// TwinCAT 3 PLC project PLC
// ProgramVersion: 3.1.4024.0
// libraries:
//   Tc2_Standard, * (Beckhoff Automation GmbH)
//   Tc2_System, * (Beckhoff Automation GmbH)
//   Tc3_Module, * (Beckhoff Automation GmbH)
//   Util, * (System)
// project tree:
//   Diagnostic/ GVL_Diagnostic.TcGVL, ST_Diagnostic.TcDUT
//   FSM/Coordinator/Enums/ E_FSM_Step.TcTLEO
//   FSM/Coordinator/FBs/ FB_FSM.TcPOU, FB_FSM_Diagnostic.TcPOU, FB_FSM_ReadCmd.TcPOU, FB_FSM_ReadCtrl.TcPOU, FB_FSM_ReadInputs.TcPOU, FB_FSM_WriteOutputs.TcPOU
//   FSM/Coordinator/ FB_FSM_Main.TcPOU
//   FSM/Coordinator/FCs/ FC_AllError.TcPOU, FC_AllStopped.TcPOU
//   FSM/Coordinator/Structs/ ST_FSM_Cmd.TcDUT, ST_FSM_Ctrl.TcDUT, ST_FSM_In.TcDUT, ST_FSM_Out.TcDUT, ST_FSM_Params.TcDUT, ST_FSM_RawIn.TcDUT, ST_FSM_RawOut.TcDUT, ST_FSM_Status.TcDUT
//   FSM/Z1/ E_Z1_Step.TcTLEO, FB_Z1_FSM.TcPOU, ST_Z1_Params.TcDUT, ST_Z1_Status.TcDUT
//   FSM/Z2/ E_Z2_Step.TcTLEO, FB_Z2_FSM.TcPOU, ST_Z2_Params.TcDUT, ST_Z2_Status.TcDUT
//   FSM/Z3/ E_Z3_Step.TcTLEO, FB_Z3_FSM.TcPOU, ST_Z3_Params.TcDUT, ST_Z3_Status.TcDUT
//   FSM/Z4/ E_Z4_Step.TcTLEO, FB_Z4_FSM.TcPOU, ST_Z4_Params.TcDUT, ST_Z4_Status.TcDUT
//   FSM/Z5/ E_Z5_Step.TcTLEO, FB_Z5_FSM.TcPOU, ST_Z5_Params.TcDUT, ST_Z5_Status.TcDUT
//   FSM/Z6/ E_Z6_Step.TcTLEO, FB_Z6_FSM.TcPOU, ST_Z6_Params.TcDUT, ST_Z6_Status.TcDUT
//   / PlcTask.TcTTO (not stored)
//   POUs/ MAIN.TcPOU
// real-time tasks:
//   TASK PlcTask: cycle T#10ms, priority 20, ADS port 350
// motion (NC):
// I/O:
//   DEVICE Dispositivo 1 (EtherCAT)
//   DEVICE Dispositivo 4 (EtherCAT), AmsNetId 5.85.198.60.5.1
//     Terminale 10 (EK1100)
// variable links:
//   PLC Instance <-> Device 4 (EtherCAT)/Term 10 (EK1100)/Term 11 (EL1809)
//     PlcTask Inputs/MAIN.stRawIn.bAckButton <-> Channel 12/Input
//     PlcTask Inputs/MAIN.stRawIn.bEmergency <-> Channel 13/Input
//     PlcTask Inputs/MAIN.stRawIn.bI{1..9} <-> Channel {1..9}/Input  (9 links)
//     PlcTask Inputs/MAIN.stRawIn.bStartButton <-> Channel 10/Input
//     PlcTask Inputs/MAIN.stRawIn.bStopButton <-> Channel 11/Input
//   PLC Instance <-> Device 4 (EtherCAT)/Term 10 (EK1100)/Term 12 (EL2809)
//     PlcTask Outputs/MAIN.stRawOut.bGreen <-> Channel 11/Output
//     PlcTask Outputs/MAIN.stRawOut.bQ{1..10} <-> Channel {1..10}/Output  (10 links)
//     PlcTask Outputs/MAIN.stRawOut.bRed <-> Channel 12/Output
//     PlcTask Outputs/MAIN.stRawOut.bYellow <-> Channel 13/Output

// ---- Diagnostic/ST_Diagnostic.TcDUT
TYPE ST_Diagnostic :
STRUCT
	aCritical : ARRAY[0..GVL_Diagnostic.cMAXEVENTS - 1] OF BOOL;	// eventi critici
	aError : ARRAY[0..GVL_Diagnostic.cMAXEVENTS - 1] OF BOOL;		// errori
	aWarning : ARRAY[0..GVL_Diagnostic.cMAXEVENTS - 1] OF BOOL;		// segnalazioni
	aInfo : ARRAY[0..GVL_Diagnostic.cMAXEVENTS - 1] OF BOOL;		// informazioni
	aVerbose : ARRAY[0..GVL_Diagnostic.cMAXEVENTS - 1] OF BOOL;		// messaggi
END_STRUCT
END_TYPE

// ---- FSM/Coordinator/Enums/E_FSM_Step.TcTLEO
{attribute 'qualified_only'}
{attribute 'strict'}
TYPE E_FSM_Step :
(
	(* special steps *)
	NoStep := -32767,		// nessuno step
	Unknown := -32000,		// step sconosciuto
	
	(* Error steps *)
	NeOrError := -990,		// non abilitata o in errore
	Recovering := -980,		// azzeramento errori

	(* Stop *)
	Stop := 0,				// stop
	
	(* Cycle *)
	Running := 100,			// funzionamento nominale delle zone
		
	(* Stopping *)
	Stopping := 900			// fase di arresto
);
END_TYPE
//  NoStep = '-32767'
//  Unknown = '-32000'
//  NeOrError = '-990'
//  Recovering = '-980'

// ---- FSM/Coordinator/Structs/ST_FSM_Cmd.TcDUT
TYPE ST_FSM_Cmd :
STRUCT
	bAck				:	BOOL;	(* Riconoscimento allarmi *)
	bStop				:	BOOL;	(* Arresta la macchina *)
	bStart				:	BOOL;	(* Mette in marcia la macchina *)
END_STRUCT
END_TYPE

// ---- FSM/Coordinator/Structs/ST_FSM_Ctrl.TcDUT
TYPE ST_FSM_Ctrl :
STRUCT
	bEmergency	:	BOOL;		// Emergenza. Deve essere TRUE perchè la macchina possa operare
	bEnable		:	BOOL;		// Abilitazione macchina. Deve essere TRUE perchè la macchina possa operare
END_STRUCT
END_TYPE

// ---- FSM/Coordinator/Structs/ST_FSM_In.TcDUT
TYPE ST_FSM_In :
STRUCT
	(* digital *)
	bEmergency		:	BOOL;				// emergenza (NC)
	bStartButton	:	BOOL;				// pulsante di start (NO)
	bStopButton		:	BOOL;				// pulsante di stop (NO)
	bAckButton		:	BOOL;				// pulsante di riconoscimento allarmi (NO)
	bI1				:	BOOL;				// Fine corsa anteriore slider 1 (NO)
	bI2				:	BOOL;				// Fine corsa posteriore slider 1 (NO)
	bI3				:	BOOL;				// Fine corsa anteriore slider 2 (NO)
	bI4				:	BOOL;				// Fine corsa posteriore slider 2 (NO)
	bI5				:	BOOL;				// Sensore ingresso slider 1 (NO)
	bI6				:	BOOL;				// Sensore presenza pezzo sotto la fresa (NO)	
	bI7				:	BOOL;				// Sensore presenza pezzo su nastro caricamento (ingresso) (NO)
	bI8				:	BOOL;				// Sensore presenza pezzo sotto il trapano (NO)
	bI9				:	BOOL;				// Sensore presenza pezzo su nastro di uscita (NO)
	
	(* analog *)

	
END_STRUCT
END_TYPE

// ---- FSM/Coordinator/Structs/ST_FSM_Out.TcDUT
TYPE ST_FSM_Out :
STRUCT
	bFixedYellow	:	BOOL;		// luce gialla fissa
	bBlinkingYellow	:	BOOL;		// luce gialla lampeggiante
	bFixedGreen		:	BOOL;		// luce verde fissa
	bBlinkingGreen	:	BOOL;		// luce verde lampeggiante	
	bFixedRed		:	BOOL;		// luce rossa fissa
	bBlinkingRed	:	BOOL;		// luce rossa lampeggiante	
	bQ1				:	BOOL;		// Rientro slider 1
	bQ2				:	BOOL;		// Estensione slider 1
	bQ3				:	BOOL;		// Rientro slider 2
	bQ4				:	BOOL;		// Estensione slider 2
	bQ5				:	BOOL;		// Motore nastro caricamento (ingresso zona Z1)
	bQ6				:	BOOL;		// Motore nastro zona fresa (Z3)
	bQ7				:	BOOL;		// Motore fresa
	bQ8				:	BOOL;		// Motore nastro zona trapano (Z4)
	bQ9				:	BOOL;		// Motore trapano
	bQ10			:	BOOL;		// Motore nastro scarico (uscita zona Z6)	
		
END_STRUCT
END_TYPE

// ---- FSM/Coordinator/Structs/ST_FSM_Params.TcDUT
TYPE ST_FSM_Params :
STRUCT
	tStoppingDelay	:	TIME	:=	T#2S;
END_STRUCT
END_TYPE

// ---- FSM/Coordinator/Structs/ST_FSM_RawIn.TcDUT
TYPE ST_FSM_RawIn :
STRUCT
	(* digital *)
	bEmergency		AT %I*	:	BOOL;		// emergenza (NC)
	bStartButton	AT %I*	:	BOOL;		// pulsante di start (NO)
	bStopButton		AT %I*	:	BOOL;		// pulsante di stop (NC)
	bAckButton		AT %I*	:	BOOL;		// pulsante di riconoscimento allarmi (NO)
	bI1				AT %I*	:	BOOL;		// Fine corsa anteriore slider 1 (NO)
	bI2				AT %I*	:	BOOL;		// Fine corsa posteriore slider 1 (NO)
	bI3				AT %I*	:	BOOL;		// Fine corsa anteriore slider 2 (NO)
	bI4				AT %I*	:	BOOL;		// Fine corsa posteriore slider 2 (NO)
	bI5				AT %I*	:	BOOL;		// Sensore ingresso slider 1 (NC)
	bI6				AT %I*	:	BOOL;		// Sensore presenza pezzo sotto la fresa (NC)	
	bI7				AT %I*	:	BOOL;		// Sensore presenza pezzo su nastro caricamento (ingresso) (NC)
	bI8				AT %I*	:	BOOL;		// Sensore presenza pezzo sotto il trapano (NC)
	bI9				AT %I*	:	BOOL;		// Sensore presenza pezzo su nastro di uscita (NC)
	
	(* analog *)

		
END_STRUCT
END_TYPE

// ---- FSM/Coordinator/Structs/ST_FSM_RawOut.TcDUT
TYPE ST_FSM_RawOut :
STRUCT
	bYellow		AT %Q*	:	BOOL;		// luce gialla
	bGreen		AT %Q*	:	BOOL;		// luce verde
	bRed		AT %Q*	:	BOOL;		// luce rossa	
	bQ1			AT %Q*	:	BOOL;		// Rientro slider 1
	bQ2			AT %Q*	:	BOOL;		// Estensione slider 1
	bQ3			AT %Q*	:	BOOL;		// Rientro slider 2
	bQ4			AT %Q*	:	BOOL;		// Estensione slider 2
	bQ5			AT %Q*	:	BOOL;		// Motore nastro caricamento (ingresso zona Z1)
	bQ6			AT %Q*	:	BOOL;		// Motore nastro zona fresa (Z3)
	bQ7			AT %Q*	:	BOOL;		// Motore fresa
	bQ8			AT %Q*	:	BOOL;		// Motore nastro zona trapano (Z4)
	bQ9			AT %Q*	:	BOOL;		// Motore trapano
	bQ10		AT %Q*	:	BOOL;		// Motore nastro scarico (uscita zona Z6)	
END_STRUCT
END_TYPE

// ---- FSM/Coordinator/Structs/ST_FSM_Status.TcDUT
TYPE ST_FSM_Status :
STRUCT
	bCritical	: BOOL;					// la macchina ha almento una condizione critica attiva
	bError		: BOOL;					// la macchina ha almento una condizione di errore attiva	
	bWarning	: BOOL;					// la macchina ha almeno una segnalazione attiva	
	bInfo		: BOOL;					// la macchina ha almeno una informazione attiva			
	bVerbose	: BOOL;					// la macchina ha almeno un messaggio attiva
	
	bFailure	: BOOL;					// la macchina è in avaria (critica + error)	
	eStep		: E_FSM_Step;			// passo della macchina a stati
	strStep		: STRING;				// passo come stringa
	tStepTime	: TIME;					// tempo di permanenza nel passo
	eErrorStep	: E_FSM_Step;			// passo in cui si è generato l'errore
	nErrorID	: DINT;					// codice di errore
	
	stZ1		: ST_Z1_Status;			// stato del dispositivo Z1
	stZ2		: ST_Z2_Status;			// stato del dispositivo Z2	
	stZ3		: ST_Z3_Status;			// stato del dispositivo Z3
	stZ4		: ST_Z4_Status;			// stato del dispositivo Z4	
	stZ5		: ST_Z5_Status;			// stato del dispositivo Z5
	stZ6		: ST_Z6_Status;			// stato del dispositivo Z6
END_STRUCT
END_TYPE

// ---- FSM/Z1/E_Z1_Step.TcTLEO
{attribute 'qualified_only'}
{attribute 'strict'}
TYPE E_Z1_Step :
(
	(* special steps *)
	NoStep := -32767,		// nessuno step
	Unknown := -32000,		// step sconosciuto
	
	(* Error steps *)
	NeOrError := -990,		// non abilitata o in errore
	Recovering := -980,		// azzeramento errori
		
	(* Stop *)
	Stop := 0,				// S0, stop
	
	(* Cycle *)
	Ready := 100,			// S1, pronto a ricevere pezzo
	DelayToFeeding := 120,	// S2, ritardo prima dell'avvio del nastro
	Loading := 140,			// S3, trasferimento pezzo verso Z2 
	DelayToZ2 := 160,		// S4, ritardo post sensore I5 verso Z2

	Done := 800,			// Ciclo concluso
	
	(* Stopping *)
	Stopping := 900	
);
END_TYPE
//  NoStep = '-32767'
//  Unknown = '-32000'
//  NeOrError = '-990'
//  Recovering = '-980'

// ---- FSM/Z1/ST_Z1_Params.TcDUT
TYPE ST_Z1_Params :
STRUCT
	tWaiting	:	TIME	:= T#3S;	// durata della fase di carico nuovo pezzo
	tTravelTime	:	TIME	:= T#4S;	// tempo per arrivare a I5
	tDelayToZ2	:	TIME	:= T#2S;	// ritardo per arrivare a Z2
	tStopDelay	:	TIME	:= T#1S;	// permanenza nello stato Stop
END_STRUCT
END_TYPE

// ---- FSM/Z1/ST_Z1_Status.TcDUT
TYPE ST_Z1_Status :
STRUCT
	eStep		:	E_Z1_Step;		// passo della macchina a stati per Z1
	strStep		:	STRING;			// passo come stringa
	tStepTime	:	TIME;			// tempo di permanenza nello stato
	eErrorStep	:	E_Z1_Step;		// stato in cui si è generato l'errore
	nErrorId	:	UDINT;			// id errore
END_STRUCT
END_TYPE

// ---- FSM/Z2/E_Z2_Step.TcTLEO
{attribute 'qualified_only'}
{attribute 'strict'}
TYPE E_Z2_Step :
(
	(* special steps *)
	NoStep := -32767,		// nessuno step
	Unknown := -32000,		// step sconosciuto
	
	(* Error steps *)
	NeOrError := -990,		// non abilitata o in errore
	Recovering := -980,		// azzeramento errori
		
	(* Stop *)
	Stop := 0,				// S0, stop
	
	(* Cycle *)
	Ready := 100,			// S1, pronto a ricevere pezzo
	WaitZ3Ready := 120,		// S2, aspetta che Z3 sia libera
	MoveForward := 140,		// S3, trasferimento pezzo verso Z2 
	MoveBackward := 160,	// S4, ritorno slitta

	Done := 800,			// Ciclo concluso
	
	(* Stopping *)
	Stopping := 900	
);
END_TYPE
//  NoStep = '-32767'
//  Unknown = '-32000'
//  NeOrError = '-990'
//  Recovering = '-980'

// ---- FSM/Z2/ST_Z2_Params.TcDUT
TYPE ST_Z2_Params :
STRUCT
	tMoving		:	TIME	:= T#6S;	// durata della fase di trasporto
	tStopDelay	:	TIME	:= T#1S;	// permanenza nello stato Stop
END_STRUCT
END_TYPE

// ---- FSM/Z2/ST_Z2_Status.TcDUT
TYPE ST_Z2_Status :
STRUCT
	eStep		:	E_Z2_Step;		// passo della macchina a stati per Z2
	strStep		:	STRING;			// passo come stringa
	tStepTime	:	TIME;			// tempo di permanenza nello stato
	eErrorStep	:	E_Z2_Step;		// stato in cui si è generato l'errore
	nErrorId	:	UDINT;			// id errore
	
END_STRUCT
END_TYPE

// ---- FSM/Z3/E_Z3_Step.TcTLEO
{attribute 'qualified_only'}
{attribute 'strict'}
TYPE E_Z3_Step :
(
	(* special steps *)
	NoStep := -32767,		// nessuno step
	Unknown := -32000,		// step sconosciuto
	
	(* Error steps *)
	NeOrError := -990,		// non abilitata o in errore
	Recovering := -980,		// azzeramento errori
		
	(* Stop *)
	Stop := 0,				// S0, stop
	
	(* Cycle *)
	Ready := 100,			// S1, pronto a ricevere pezzo
	MoveToMill := 120,		// S2, avanza il nastro fino alla fresa
	Milling := 140,			// S3, lavorazione con la fresa
	WaitZ4Ready := 160,		// S4, attende che Z4 sia ready
	MoveToZ4 := 180,		// S5, avanza il nastro fino a Z4

	Done := 800,			// Ciclo concluso
	
	(* Stopping *)
	Stopping := 900	
);
END_TYPE
//  NoStep = '-32767'
//  Unknown = '-32000'
//  NeOrError = '-990'
//  Recovering = '-980'

// ---- FSM/Z3/ST_Z3_Params.TcDUT
TYPE ST_Z3_Params :
STRUCT
	tMilling	:	TIME	:= T#6S;	// durata della fase di fresatura
	tDelayToZ4	:	TIME	:= T#3S;	// ritardo per arrivare a Z4
	tStopDelay	:	TIME	:= T#1S;	// permanenza nello stato Stop
	tRecovering	: TIME		:= T#2S; 	// tempo di uscita dallo stato di Recovering
END_STRUCT
END_TYPE

// ---- FSM/Z3/ST_Z3_Status.TcDUT
TYPE ST_Z3_Status :
STRUCT
	eStep		:	E_Z3_Step;		// passo della macchina a stati per Z3
	strStep		:	STRING;			// passo come stringa
	tStepTime	:	TIME;			// tempo di permanenza nello stato
	eErrorStep	:	E_Z3_Step;		// stato in cui si è generato l'errore
	nErrorId	:	UDINT;			// id errore
END_STRUCT
END_TYPE

// ---- FSM/Z4/E_Z4_Step.TcTLEO
{attribute 'qualified_only'}
{attribute 'strict'}
TYPE E_Z4_Step :
(
	(* special steps *)
	NoStep := -32767,		// nessuno step
	Unknown := -32000,		// step sconosciuto
	
	(* Error steps *)
	NeOrError := -990,		// non abilitata o in errore
	Recovering := -980,		// azzeramento errori
		
	(* Stop *)
	Stop := 0,				// S0, stop
	
	(* Cycle *)
	Ready := 100,			// S1, pronto a ricevere pezzo
	MoveToDrill := 120,		// S2, avanza il nastro fino al trapano
	Drilling := 140,		// S3, lavorazione con il trapano
	WaitZ5Ready := 160,		// S4, attende che Z5 sia ready
	MoveToZ5 := 180,		// S5, avanza il nastro fino a Z5

	Done := 800,			// Ciclo concluso
	
	(* Stopping *)
	Stopping := 900	
);
END_TYPE
//  NoStep = '-32767'
//  Unknown = '-32000'
//  NeOrError = '-990'
//  Recovering = '-980'

// ---- FSM/Z4/ST_Z4_Params.TcDUT
TYPE ST_Z4_Params :
STRUCT
	tDrilling	:	TIME	:= T#4S;	// durata della fase di foratura
	tDelayToZ5	:	TIME	:= T#1S;	// ritardo per arrivare a Z5
	tStopDelay	:	TIME	:= T#1S;	// permanenza nello stato Stop
	tRecovering :   TIME	:= T#2S;
END_STRUCT
END_TYPE

// ---- FSM/Z4/ST_Z4_Status.TcDUT
TYPE ST_Z4_Status :
STRUCT
	eStep		:	E_Z4_Step;		// passo della macchina a stati per Z4
	strStep		:	STRING;			// passo come stringa
	tStepTime	:	TIME;			// tempo di permanenza nello stato
	eErrorStep	:	E_Z4_Step;		// stato in cui si è generato l'errore
	nErrorId	:	UDINT;			// id errore
END_STRUCT
END_TYPE

// ---- FSM/Z5/E_Z5_Step.TcTLEO
{attribute 'qualified_only'}
{attribute 'strict'}
TYPE E_Z5_Step :
(
	(* special steps *)
	NoStep := -32767,		// nessuno step
	Unknown := -32000,		// step sconosciuto
	
	(* Error steps *)
	NeOrError := -990,		// non abilitata o in errore
	Recovering := -980,		// azzeramento errori
		
	(* Stop *)
	Stop := 0,				// S0, stop
	
	(* Cycle *)
	Ready := 100,			// S1, pronto a ricevere pezzo
	WaitZ6Ready := 120,		// S2, aspetta che Z6 sia libera
	MoveForward := 140,		// S3, trasferimento pezzo verso Z6 
	MoveBackward := 160,	// S4, ritorno slitta

	Done := 800,			// Ciclo concluso
	
	(* Stopping *)
	Stopping := 900	
);
END_TYPE
//  NoStep = '-32767'
//  Unknown = '-32000'
//  NeOrError = '-990'
//  Recovering = '-980'

// ---- FSM/Z5/ST_Z5_Params.TcDUT
TYPE ST_Z5_Params :
STRUCT
	tMoving		:	TIME	:= T#6S;	// durata della fase di trasporto
	tStopDelay	:	TIME	:= T#1S;	// permanenza nello stato Stop
END_STRUCT
END_TYPE

// ---- FSM/Z5/ST_Z5_Status.TcDUT
TYPE ST_Z5_Status :
STRUCT
	eStep		:	E_Z5_Step;		// passo della macchina a stati per Z5
	strStep		:	STRING;			// passo come stringa
	tStepTime	:	TIME;			// tempo di permanenza nello stato
	eErrorStep	:	E_Z5_Step;		// stato in cui si è generato l'errore
	nErrorId	:	UDINT;			// id errore
END_STRUCT
END_TYPE

// ---- FSM/Z6/E_Z6_Step.TcTLEO
{attribute 'qualified_only'}
{attribute 'strict'}
TYPE E_Z6_Step :
(
	(* special steps *)
	NoStep := -32767,		// nessuno step
	Unknown := -32000,		// step sconosciuto
	
	(* Error steps *)
	NeOrError := -990,		// non abilitata o in errore
	Recovering := -980,		// azzeramento errori
		
	(* Stop *)
	Stop := 0,				// S0, stop
	
	(* Cycle *)
	Ready := 100,			// S1, pronto a ricevere pezzo
	Loading := 120,			// S2, trasferimento pezzo verso I9
	WaitUnloading := 140,	// S3, attesa rimozione pezzo da piattaforma scarico 

	Done := 800,			// Ciclo concluso
	
	(* Stopping *)
	Stopping := 900	
);
END_TYPE
//  NoStep = '-32767'
//  Unknown = '-32000'
//  NeOrError = '-990'
//  Recovering = '-980'

// ---- FSM/Z6/ST_Z6_Params.TcDUT
TYPE ST_Z6_Params :
STRUCT
	tDelayToEnd	:	TIME	:= T#2S;	// ritardo per arrivare a fine nastro
	tUnloading	:	TIME	:= T#3S;	// durata della fase di scarico
	tStopDelay	:	TIME	:= T#1S;	// permanenza nello stato Stop
END_STRUCT
END_TYPE

// ---- FSM/Z6/ST_Z6_Status.TcDUT
TYPE ST_Z6_Status :
STRUCT
	eStep		:	E_Z6_Step;		// passo della macchina a stati per Z6
	strStep		:	STRING;			// passo come stringa
	tStepTime	:	TIME;			// tempo di permanenza nello stato
	eErrorStep	:	E_Z6_Step;		// stato in cui si è generato l'errore
	nErrorId	:	UDINT;			// id errore
END_STRUCT
END_TYPE

// ---- Diagnostic/GVL_Diagnostic.TcGVL
{attribute 'qualified_only'}
VAR_GLOBAL CONSTANT
	cMAXEVENTS : UDINT := 64;
END_VAR

// ---- FSM/Coordinator/FBs/FB_FSM.TcPOU
FUNCTION_BLOCK FB_FSM
VAR_INPUT
	stIn		:	ST_FSM_In;
	stCtrl		:	ST_FSM_Ctrl;
	stCmd		:	ST_FSM_Cmd;
	stParams	:	ST_FSM_Params;
END_VAR
VAR_IN_OUT
	stStatus	:	ST_FSM_Status;	
END_VAR
VAR_OUTPUT	
	eStep		:	E_FSM_Step;
	tStepTime	:	TIME;
	eErrStep	:	E_FSM_Step;
	nErrId		:	DINT;
	// Digital Outputs
	stOut		:	ST_FSM_Out;	
	
END_VAR
VAR
	// FSM internal variables
	bInitialized	:	BOOL;
	eNewstep		:	E_FSM_Step;
	bEntryact		:	BOOL;
	fbTonStep		:	TON;

	(* filters on other input from plant *)
	
	(* stop request *)	
	bStopRequest	:	BOOL;
	
	// all zones are stopped
	bAllZoneStopped	:	BOOL;	
END_VAR

IF NOT bInitialized THEN
	(* here you can wait events from other controllers *)
	eNewStep := E_FSM_Step.NoStep;
	stStatus.eStep := E_FSM_Step.NeOrError;
	bEntryact := FALSE;
	bInitialized := TRUE;
ELSE
	// --- FSM Cyclical Code ----------------------------------------------
	
	// update of the enabling conditions (bStop, alarms, etc.)
	
	// 1. FSM Preamble ----------------------------------------------------
    // 1.a State machine disabled or failure
	IF NOT stCtrl.bEnable OR NOT stCtrl.bEmergency OR stStatus.bFailure THEN
		eNewStep := E_FSM_Step.NeOrError;
	END_IF

	// 1.b Update eStep with the required step to perform
	//     and set bEntryact to FALSE in order to enable the Entry action
	IF eNewstep <> E_FSM_Step.NoStep THEN
		stStatus.eStep := eNewstep;
		eNewstep := E_FSM_Step.NoStep;
		bEntryact := FALSE;
	END_IF;	
	
	// 1.c Do filters on signals	

	
	// Do requests, for example to stop the machine
	IF stCmd.bStop THEN
		bStopRequest := TRUE;
	END_IF

	// 2. The main switch-case ---------------------------------------------------
	CASE stStatus.eStep OF
    E_FSM_Step.NeOrError :
			// on entry action
			IF NOT bEntryact THEN
				stStatus.bFailure := TRUE;
				bEntryact := TRUE;
			END_IF
			
			// body
			stOut.bFixedGreen := TRUE;
			stOut.bBlinkingGreen := FALSE;
			stOut.bFixedRed := FALSE;
			stOut.bBlinkingRed := FALSE;
			stOut.bFixedYellow := FALSE;
			stOut.bBlinkingYellow := FALSE;
					
			
			// next state transition
			IF stCtrl.bEnable THEN
				IF stCmd.bAck THEN
					eNewStep := E_Z3_Step.Recovering;
				END_IF
			END_IF
		
			// on exit action
			IF eNewStep <> E_Z3_Step.NoStep THEN
				nErrId := 0;
				eErrStep := E_Z3_Step.NoStep;
			END_IF
						
	ELSE
		// this happens also if we forget to code one step 
		eNewstep := E_FSM_Step.NeOrError;
		stStatus.eErrorStep := E_FSM_Step.Unknown;
		stStatus.nErrorID := -9;
	END_CASE;
	
	// 3. FSM Epilogue ------------------------------------------------------
	
	// Elapsed time into the current step
	fbTonStep(IN := (eNewstep = E_FSM_Step.NoStep), PT := T#500H );
	stStatus.tStepTime := fbTonStep.ET;
	
END_IF

END_FUNCTION_BLOCK

// ---- FSM/Coordinator/FBs/FB_FSM_Diagnostic.TcPOU
FUNCTION_BLOCK FB_FSM_Diagnostic
VAR_INPUT
	stIn : ST_FSM_In;
	stOut : ST_FSM_Out;
	stParams : ST_FSM_Params;
	stCtrl : ST_FSM_Ctrl;
	bHwError : BOOL;
	bAck : BOOL;
	stStatus : ST_FSM_Status;	
END_VAR
VAR_IN_OUT
END_VAR
VAR_OUTPUT
	bCritical	: BOOL;
	bError		: BOOL;
	bWarning	: BOOL;
	bInfo		: BOOL;
	bVerbose	: BOOL;
	bFailure	: BOOL;
	bBlinking	: BOOL;
	bFixed		: BOOL;
END_VAR
VAR
END_VAR

// on Ack, reset holding conditions
IF bAck THEN
	bCritical := FALSE;
	bError := FALSE;
	bWarning := FALSE;
	bInfo := FALSE;
	bVerbose := FALSE;
	bBlinking := FALSE;
END_IF

// update critical condition
bCritical := FC_AllError(stStatus) OR NOT stCtrl.bEmergency;

// update holding conditions
bFailure := bCritical OR bError;

bBlinking := bFailure;
bFixed := bWarning;

END_FUNCTION_BLOCK

// ---- FSM/Coordinator/FCs/FC_AllError.TcPOU
FUNCTION FC_AllError : BOOL
VAR_INPUT
	stStatus	:	ST_FSM_Status;
END_VAR
VAR
END_VAR

FC_AllError := (stStatus.stZ1.eStep = E_Z1_Step.NeOrError) AND
                 (stStatus.stZ2.eStep = E_Z2_Step.NeOrError) AND
                 (stStatus.stZ3.eStep = E_Z3_Step.NeOrError) AND	
                 (stStatus.stZ4.eStep = E_Z4_Step.NeOrError) AND
                 (stStatus.stZ5.eStep = E_Z5_Step.NeOrError) AND	
                 (stStatus.stZ6.eStep = E_Z6_Step.NeOrError);

END_FUNCTION

// ---- FSM/Coordinator/FBs/FB_FSM_ReadCmd.TcPOU
FUNCTION_BLOCK FB_FSM_ReadCmd
VAR_INPUT
	stIn	:	ST_FSM_In;
END_VAR
VAR_OUTPUT
	stCmd	:	ST_FSM_Cmd;
END_VAR
VAR
	fbTpStart	: TP;
	fbTpStop	: TP;	
	fbTpAck		: TP;
END_VAR

// filters on input button
fbTpStart( IN := stIn.bStartButton, PT := T#50MS );
fbTpStop( IN := stIn.bStopButton, PT := T#50MS );
fbTpAck( IN := stIn.bAckButton, PT := T#50MS );

stCmd.bStart	:= fbTpStart.Q;
stCmd.bStop		:= fbTpStop.Q;
stCmd.bAck		:= fbTpAck.Q;

END_FUNCTION_BLOCK

// ---- FSM/Coordinator/FBs/FB_FSM_ReadCtrl.TcPOU
FUNCTION_BLOCK FB_FSM_ReadCtrl
VAR_INPUT
	nId:	INT;
	bEnable : BOOL;
	stIn : ST_FSM_In;
END_VAR
VAR_OUTPUT
	stCtrl : ST_FSM_Ctrl;
END_VAR
VAR
	fbTonStartup: TON;
END_VAR

fbTonStartup(IN := TRUE, PT := T#3S);
stCtrl.bEmergency := stIn.bEmergency;
stCtrl.bEnable := fbTonStartup.Q AND bEnable;

END_FUNCTION_BLOCK

// ---- FSM/Coordinator/FBs/FB_FSM_ReadInputs.TcPOU
FUNCTION_BLOCK FB_FSM_ReadInputs
VAR_INPUT
END_VAR
VAR_IN_OUT
	stRawIn		:	ST_FSM_RawIn;
END_VAR
VAR_OUTPUT
	stIn		:	ST_FSM_In;
END_VAR
VAR
END_VAR

// digital inputs
stIn.bEmergency := stRawIn.bEmergency;   // NOTA: Emg è sempre attivo basso
stIn.bStartButton := stRawIn.bStartButton;
stIn.bStopButton := NOT stRawIn.bStopButton;
stIn.bAckButton := stRawIn.bAckButton;
stIn.bI1 := stRawIn.bI1;
stIn.bI2 := stRawIn.bI2;
stIn.bI3 := stRawIn.bI3;
stIn.bI4 := stRawIn.bI4;
stIn.bI5 := NOT stRawIn.bI5;
stIn.bI6 := NOT stRawIn.bI6;
stIn.bI7 := NOT stRawIn.bI7;
stIn.bI8 := NOT stRawIn.bI8;
stIn.bI9 := NOT stRawIn.bI9;

END_FUNCTION_BLOCK

// ---- FSM/Coordinator/FBs/FB_FSM_WriteOutputs.TcPOU
FUNCTION_BLOCK FB_FSM_WriteOutputs
VAR_INPUT
	stOut		:	ST_FSM_Out;
END_VAR
VAR_OUTPUT
	stRawOut	:	ST_FSM_RawOut;
END_VAR
VAR
	fbBlink		:	BLINK;
END_VAR

// blinking
fbBlink(ENABLE:= TRUE, TIMELOW:= T#500MS, TIMEHIGH:= T#500MS);

// indicators on control panel
IF stOut.bBlinkingYellow THEN
	stRawOut.bYellow := fbBlink.OUT;
ELSE
	IF stOut.bFixedYellow THEN
		stRawOut.bYellow := TRUE;
	ELSE
		stRawOut.bYellow := FALSE;		
	END_IF
END_IF

IF stOut.bBlinkingGreen THEN
	stRawOut.bGreen := fbBlink.OUT;
ELSE
	IF stOut.bFixedGreen THEN
		stRawOut.bGreen := TRUE;
	ELSE
		stRawOut.bGreen := FALSE;		
	END_IF
END_IF

IF stOut.bBlinkingRed THEN
	stRawOut.bRed := fbBlink.OUT;
ELSE
	IF stOut.bFixedRed THEN
		stRawOut.bRed := TRUE;
	ELSE
		stRawOut.bRed := FALSE;		
	END_IF
END_IF


// other digital outputs
stRawOut.bQ1 := stOut.bQ1;
stRawOut.bQ2 := stOut.bQ2;
stRawOut.bQ3 := stOut.bQ3;
stRawOut.bQ4 := stOut.bQ4;
stRawOut.bQ5 := stOut.bQ5;
stRawOut.bQ6 := stOut.bQ6;
stRawOut.bQ7 := stOut.bQ7;
stRawOut.bQ8 := stOut.bQ8;
stRawOut.bQ9 := stOut.bQ9;
stRawOut.bQ10 := stOut.bQ10;

END_FUNCTION_BLOCK

// ---- FSM/Coordinator/FB_FSM_Main.TcPOU
FUNCTION_BLOCK FB_FSM_Main
VAR_INPUT
	(* main inputs to the state machine *)
	bEnable			: BOOL;		// state machine enable
	tTaskCycleTime	: UDINT;
	nId				: USINT;	
	bHwError		: BOOL;
END_VAR
VAR_OUTPUT
END_VAR
VAR_IN_OUT
	(* machine I/Os *)
	stRawIn		:	ST_FSM_RawIn;
	stIn		:	ST_FSM_In;
	stRawOut	:	ST_FSM_RawOut;
	stOut		:	ST_FSM_Out;
	stCtrl		:	ST_FSM_Ctrl;
	
	(* state machine internals, useful for debugging  *)
	stStatus	:	ST_FSM_Status;	
END_VAR
VAR
	bInitialized	: 	BOOL;		// FB initialization
	stCmd			:	ST_FSM_Cmd;
	stParams		:	ST_FSM_Params;	
	errno			:	INT;
	fbReadCmd		:	FB_FSM_ReadCmd;
	fbReadCtrl		:	FB_FSM_ReadCtrl;
	fbReadIn		:	FB_FSM_ReadInputs;
	fbDiagnostic	:	FB_FSM_Diagnostic;
	fbWriteOut		:	FB_FSM_WriteOutputs;
	
	(* instantiate the coordinator state machine *)
    fbStateMachine	:	FB_FSM;
	
	(* zone parameters *)
	stZ1Params		:	ST_Z1_Params;
	stZ2Params		:	ST_Z2_Params;
	stZ3Params		:	ST_Z3_Params;	
	stZ4Params		:	ST_Z4_Params;	
	stZ5Params		:	ST_Z5_Params;	
	stZ6Params		:	ST_Z6_Params;	
	
	(* instantiate the six zone state machines *)
	// to be done...
	fbZ1Machine		:	FB_Z1_FSM;
	fbZ2Machine		:	FB_Z2_FSM;
	fbZ3Machine		:	FB_Z3_FSM;
	fbZ4Machine		:	FB_Z4_FSM;
	fbZ5Machine		:	FB_Z5_FSM;
	fbZ6Machine		:	FB_Z6_FSM;
	
END_VAR

IF NOT bInitialized THEN
	// start-up operations
	bInitialized := TRUE;
ELSE
// 01. Read inputs, controls, parameters and commands
	fbReadIn(stRawIn := stRawIn,
             stIn => stIn);	
	fbReadCtrl(nId := nId,
               bEnable := bEnable,
               stIn := stIn,
               stCtrl => stCtrl);
    fbReadCmd(stIn := stIn,
              stCmd => stCmd);

	// 02. events management fbDiagnostic
	fbDiagnostic(
	stIn:= stIn, 
	stOut:= stOut, 
	stParams:= stParams, 
	stCtrl:= stCtrl, 
	bHwError:= bHwError, 
	bAck:= stCmd.bAck, 
	stStatus:= stStatus);
	
	stStatus.bCritical := fbDiagnostic.bCritical;
	stStatus.bError := fbDiagnostic.bError;
	stStatus.bWarning := fbDiagnostic.bWarning;
	stStatus.bInfo := fbDiagnostic.bInfo;
	stStatus.bVerbose := fbDiagnostic.bVerbose;
	stStatus.bFailure := fbDiagnostic.bFailure;
	stOut.bBlinkingRed := fbDiagnostic.bCritical;
	stOut.bBlinkingYellow := fbDiagnostic.bBlinking;
	stOut.bFixedYellow := fbDiagnostic.bFixed;	

	(* 03. call the coordinator state machine *)
    fbStateMachine( stIn := stIn,
                    stCtrl := stCtrl,
                    stCmd := stCmd,
                    stParams := stParams,
                    stStatus := stStatus);
	 
    (* 04. six secondary state machines  *)
	
	(* call Z1 state machine  *)
	fbZ1Machine(
		bEnable:= NOT(stStatus.bFailure), 
		bAck:= (stStatus.eStep = E_FSM_Step.Recovering), 
		bStart:= (stStatus.eStep = E_FSM_Step.Running), 
		bStop:= (stStatus.eStep = E_FSM_Step.Stopping), 
		bI5:= stIn.bI5, 
		bI7:= stIn.bI7, 
		stParams:= stZ1Params, 
		stStatus:= stStatus, 
		bQ5=> stOut.bQ5);
	
	(* call Z2 state machine  *)
	fbZ2Machine(
		bEnable:= NOT(stStatus.bFailure), 
		bAck:= (stStatus.eStep = E_FSM_Step.Recovering), 
		bStop:= (stStatus.eStep = E_FSM_Step.Stopping), 
		bI1:= stIn.bI1, 
		bI2:= stIn.bI2, 
		stParams:= stZ2Params, 
		stStatus:= stStatus, 
		bQ1=> stOut.bQ1, 
		bQ2=> stOut.bQ2);
	
	(* call Z3 state machine  *)	
	fbZ3Machine(
		bEnable:= NOT(stStatus.bFailure), 
		bAck:= (stStatus.eStep = E_FSM_Step.Recovering), 
		bStop:= (stStatus.eStep = E_FSM_Step.Stopping), 
		bI6:= stIn.bI6, 
		stParams:= stZ3Params, 
		stStatus:= stStatus, 
		bQ6=> stOut.bQ6, 
		bQ7=> stOut.bQ7);
	
	(* call Z4 state machine  *)	
	fbZ4Machine(
		bEnable:= NOT(stStatus.bFailure), 
		bAck:= (stStatus.eStep = E_FSM_Step.Recovering), 
		bStop:= (stStatus.eStep = E_FSM_Step.Stopping), 
		bI8:= stIn.bI8, 
		stParams:= stZ4Params, 
		stStatus:= stStatus, 
		bQ8=> stOut.bQ8, 
		bQ9=> stOut.bQ9);	
	
	(* call Z5 state machine  *)
	fbZ5Machine(
		bEnable:= NOT(stStatus.bFailure), 
		bAck:= (stStatus.eStep = E_FSM_Step.Recovering), 
		bStop:= (stStatus.eStep = E_FSM_Step.Stopping), 
		bI3:= stIn.bI3, 
		bI4:= stIn.bI4, 
		stParams:= stZ5Params, 
		stStatus:= stStatus, 
		bQ3=> stOut.bQ3, 
		bQ4=> stOut.bQ4);		
	
	(* call Z6 state machine  *)
	fbZ6Machine(
		bEnable:= NOT(stStatus.bFailure), 
		bAck:= (stStatus.eStep = E_FSM_Step.Recovering), 
		bStop:= (stStatus.eStep = E_FSM_Step.Stopping), 
		bI9:= stIn.bI9, 
		stParams:= stZ6Params, 
		stStatus:= stStatus, 
		bQ10=> stOut.bQ10);	
		
	
	// 05. write outputs and machine information
	fbWriteOut( stOut:= stOut, 
				stRawOut => stRawOut);
				
	// 06. end - other operations			 
END_IF

END_FUNCTION_BLOCK

// ---- FSM/Z1/FB_Z1_FSM.TcPOU
FUNCTION_BLOCK FB_Z1_FSM
VAR_INPUT
	bEnable		:	BOOL;
	bAck		:	BOOL;
	bStart		:	BOOL;
	bStop		:	BOOL;
	bI5			:	BOOL;
	bI7			:	BOOL;
	stParams	:	ST_Z1_Params;	
END_VAR
VAR_IN_OUT
	stStatus	:	ST_FSM_Status;	
END_VAR
VAR_OUTPUT
	// Digital Outputs
	bQ5			:	BOOL;	
	bErr		:	BOOL;
END_VAR
VAR
	// FSM internal variables
	bInitialized	:	BOOL;
	eNewstep		:	E_Z1_Step;
	bEntryact		:	BOOL;
	fbTonStep		:	TON;
	
	fbRtStart		:	R_TRIG;
	fbRtStop		:	R_TRIG;
	fbRtI5			:	R_TRIG;
	fbRtI7			:	R_TRIG;
	bStopRequest	:	BOOL;


END_VAR

IF NOT bInitialized THEN
	eNewstep :=  E_Z1_Step.NoStep;
	stStatus.stZ1.eStep :=  E_Z1_Step.NeOrError;
	bEntryact := FALSE;
	bInitialized := TRUE;	
	bErr := FALSE;
	stStatus.stZ1.eErrorStep :=  E_Z1_Step.NoStep;	
	stStatus.stZ1.nErrorId := 0;	
ELSE
	(* fronti *)
	fbRtStart(CLK:= bStart);
	fbRtStop(CLK:= bStop);	
	fbRtI5(CLK := bI5);
	fbRtI7(CLK := bI7);
	
	(* richieste *)
	IF fbRtStop.Q THEN
		bStopRequest := TRUE;
	END_IF; 

	(* disabilitata o avaria *)
	IF NOT bEnable THEN
		eNewstep := E_Z1_Step.NeOrError;
	END_IF;
	
	(* aggiornamento dello stato *)
	IF eNewstep <>  E_Z1_Step.NoStep THEN
		stStatus.stZ1.eStep := eNewstep;
		eNewstep :=  E_Z1_Step.NoStep;
		bEntryact := FALSE;
	END_IF;	
	
	(* switch - case della MSF *)
	CASE stStatus.stZ1.eStep OF
		
	// NeOrError ---------------------------------
	E_Z1_Step.NeOrError :
			// on entry action
			IF NOT bEntryact THEN
				bErr := TRUE;
				bEntryact := TRUE;
			END_IF
			
			// body
			bErr := TRUE;
					
			
			// next state transition
			IF bEnable THEN
				IF bAck THEN
					eNewStep := E_Z1_Step.Recovering;
				END_IF
			END_IF
		
			// on exit action
			IF eNewStep <> E_Z1_Step.NoStep THEN
				stStatus.stZ1.nErrorId := 1;
				stStatus.stZ1.eErrorStep := E_Z1_Step.NoStep;
			END_IF	
	E_Z1_Step.Stop :
		// on entry action
		IF NOT bEntryact THEN
			bErr := FALSE;
			bStopRequest := FALSE;
			bEntryact := TRUE;
		END_IF
		
		// body
		bQ5 := FALSE;
		
		// next state transition
		IF (stStatus.stZ1.tStepTime > stParams.tStopDelay AND fbRtStart.Q) THEN
			eNewStep := E_Z1_Step.Ready;
		END_IF
		
		// on exit action
		IF eNewStep <> E_Z1_Step.NoStep THEN
			;
		END_IF
		
	// Ready ---------------------------------	
	E_Z1_Step.Ready:
		// on entry action
		IF NOT bEntryact THEN
			bErr := FALSE;
			bEntryact := TRUE;
		END_IF
		
		// body	
		bQ5 := FALSE;
	
		// next state transition
		IF bStopRequest THEN
			eNewStep := E_Z1_Step.Stop;
		ELSE
			IF fbRtI7.Q THEN
				eNewStep := E_Z1_Step.DelayToFeeding;
			END_IF
		END_IF

		// on exit action
		IF eNewStep <> E_Z1_Step.NoStep THEN
			;
		END_IF
		
	// DelayToFeeding ---------------------------------	
	E_Z1_Step.DelayToFeeding:
		// on entry action
		IF NOT bEntryact THEN
			bErr := FALSE;
			bEntryact := TRUE;
		END_IF
		
		// body	
		bQ5 := FALSE;

		// next state transition
		IF bStopRequest THEN
			eNewStep := E_Z1_Step.Stop;
		ELSIF (stStatus.stZ1.tStepTime > stParams.tWaiting AND stStatus.stZ2.eStep=E_Z2_Step.Ready) THEN
			eNewStep := E_Z1_Step.Loading;
		END_IF

		// on exit action
		IF eNewStep <> E_Z1_Step.NoStep THEN
			;
		END_IF

	// Loading ---------------------------------	
	E_Z1_Step.Loading:
		// on entry action
		IF NOT bEntryact THEN
			bErr := FALSE;
			bEntryact := TRUE;
		END_IF
		
		// body		
		bQ5 := TRUE;

		// next state transition	
		IF (stStatus.stZ1.tStepTime < stParams.tTravelTime AND fbRtI5.Q) THEN
			eNewStep := E_Z1_Step.DelayToZ2;
		ELSIF (stStatus.stZ1.tStepTime > stParams.tTravelTime) THEN
			eNewStep := E_Z1_Step.NeOrError;
		END_IF

		// on exit action
		IF eNewStep <> E_Z1_Step.NoStep THEN
			;
		END_IF

	// DelayToZ2 ---------------------------------	
	E_Z1_Step.DelayToZ2:
		// on entry action
		IF NOT bEntryact THEN
			bErr := FALSE;
			bEntryact := TRUE;
		END_IF
		
		// body	
		bQ5 := TRUE;

		// next state transition
		IF stStatus.stZ1.tStepTime >= stParams.tTravelTime THEN
			IF NOT(bI5) THEN
				eNewStep := E_Z1_Step.Done;
			ELSE 
				eNewStep := E_Z1_Step.NeOrError;
			END_IF
		END_IF

		// on exit action
		IF eNewStep <> E_Z1_Step.NoStep THEN
			;
		END_IF

	// Done ---------------------------------		
	E_Z1_Step.Done:
		// on entry action
		IF NOT bEntryact THEN
			bErr := FALSE;
			bEntryact := TRUE;
		END_IF
		
		// body		
		bQ5 := FALSE;
		
		// next state transition
		eNewStep := E_Z1_Step.Ready;

		// on exit action
		IF eNewStep <> E_Z1_Step.NoStep THEN
			;
		END_IF

	// Recovering ---------------------------------	
	E_Z1_Step.Recovering:
		// on entry action
		IF NOT bEntryact THEN
			bErr := FALSE;
			bEntryact := TRUE;
		END_IF
		
		// body	
		bQ5 := FALSE;

		// next state transition	
		eNewStep := E_Z1_Step.Stop;

		// on exit action
		IF eNewStep <> E_Z1_Step.NoStep THEN
			;
		END_IF		

	ELSE
			eNewstep :=  E_Z1_Step.NeOrError;
			stStatus.stZ1.eErrorStep :=  E_Z1_Step.Unknown;			
			stStatus.stZ1.nErrorId := 16#0001_9999;	
	END_CASE
	
	(* call FBs *)
	
	(* tempo di permanenza nello step *)
	fbTonStep(IN := (eNewstep =  E_Z1_Step.NoStep), PT := T#500H);
	stStatus.stZ1.tStepTime := fbTonStep.ET;	
	
END_IF

END_FUNCTION_BLOCK

// ---- FSM/Z2/FB_Z2_FSM.TcPOU
FUNCTION_BLOCK FB_Z2_FSM
VAR_INPUT
	bEnable		:	BOOL;
	bAck		:	BOOL;
	bStop		:	BOOL;
	bI1			:	BOOL;
	bI2			:	BOOL;
	stParams	:	ST_Z2_Params;	
END_VAR
VAR_IN_OUT
	stStatus	:	ST_FSM_Status;	
END_VAR
VAR_OUTPUT
	// Digital Outputs
	bQ1			:	BOOL;
	bQ2			:	BOOL;	
	bErr		:	BOOL;
END_VAR
VAR
	// FSM internal variables
	bInitialized	:	BOOL;
	eNewstep		:	E_Z2_Step;
	bEntryact		:	BOOL;
	fbTonStep		:	TON;
	fbRtStop		:	R_TRIG;
	fbRtI1			:	R_TRIG;
	fbRtI2			:	R_TRIG;
	bStopRequest	:	BOOL;	
	bConveyorLoaded :   BOOL;
END_VAR

IF NOT bInitialized THEN
	eNewstep :=  E_Z2_Step.NoStep;
	stStatus.stZ2.eStep :=  E_Z2_Step.NeOrError;
	bEntryact := FALSE;
	bInitialized := TRUE;	
	bErr := FALSE;
	stStatus.stZ2.eErrorStep :=  E_Z2_Step.NoStep;	
	stStatus.stZ2.nErrorId := 0;	
ELSE
	(* fronti *)
	fbRtStop(CLK:= bStop);	
	fbRtI1(CLK := bI1);
	fbRtI2(CLK := bI2);
	
	(* richieste *)
	IF fbRtStop.Q THEN
		bStopRequest := TRUE;
	END_IF; 

	(* disabilitata o avaria *)
	IF NOT bEnable THEN
		eNewstep := E_Z2_Step.NeOrError;
	END_IF;
	
	(* aggiornamento dello stato *)
	IF eNewstep <>  E_Z2_Step.NoStep THEN
		stStatus.stZ2.eStep := eNewstep;
		eNewstep :=  E_Z2_Step.NoStep;
		bEntryact := FALSE;
	END_IF;	
	
	(* switch - case della MSF *)
	CASE stStatus.stZ2.eStep OF
		
	// NeOrError -----------------------------------------
	E_Z2_Step.NeOrError :
		// entry action
		IF NOT bEntryact THEN
			bErr := TRUE;
			bEntryact := TRUE;
		END_IF
		
		// body
		bQ1 := FALSE;
		bQ2 := FALSE;
		
		// transition from Ne0rError to Recovering
		IF (bEnable AND bAck) THEN
			eNewStep := E_Z2_Step.Recovering;
		END_IF
		
		// exit action
		IF eNewStep <> E_Z2_Step.NoStep THEN
			stStatus.stZ2.nErrorID := 2;
			stStatus.stZ2.eErrorStep := E_Z2_Step.NoStep;
		END_IF	
	
    // Recovering		
    E_Z2_Step.Recovering :
		// entry action
		IF NOT bEntryact THEN
			bErr := FALSE;
			bEntryact := TRUE;
		END_IF
		
		// body	
		bQ1 := NOT(bI2);
		bQ2 := FALSE;
		
		// transition from Recovering to Stop
		IF (fbRtI2.Q) THEN
			eNewStep := E_Z2_Step.Stop;
		END_IF
		
		// on exit action
		IF eNewStep <> E_Z2_Step.NoStep THEN
			;
		END_IF				
	
    //Stop
    E_Z2_Step.Stop :
		// entry action
		IF NOT bEntryact THEN
			bErr := FALSE;
			bStopRequest := FALSE;
			bEntryact := TRUE;
		END_IF;
		
		//body
		bQ1 := FALSE;
		bQ2 := FALSE;
		
		//transition from Stop to Ready
		IF (stStatus.stZ2.tStepTime > stParams.tStopDelay) THEN
			eNewStep := E_Z2_Step.Ready; 
		END_IF;
		
		// exit action
		IF eNewStep <> E_Z2_Step.NoStep THEN
			;
		END_IF;
			
	//Ready
	E_Z2_Step.Ready :
		// entry action
		IF NOT bEntryact THEN
			bErr := FALSE;
			bEntryact := TRUE;
		END_IF;	
		
		// body
		bQ1 :=  FALSE;
		bQ2 := FALSE;
		
		//transition from Ready to Recovering / WaitZ3Ready
		IF (bStopRequest) THEN 
			eNewStep := E_Z2_Step.Recovering;
		ELSIF stStatus.stZ1.eStep = E_Z1_Step.DelayToZ2 THEN
			eNewStep := E_Z2_Step.WaitZ3Ready;
		END_IF;
		
		// exit action 
		IF eNewStep <> E_Z2_Step.NoStep THEN
			;
		END_IF;	
	
	// WaitZ3Ready
	E_Z2_Step.WaitZ3Ready :
		// entry action
		IF NOT bEntryact THEN
			bErr := FALSE;
			bEntryact := TRUE;
		END_IF;
		
		// body
		bQ1 := FALSE;
		bQ2 := FALSE;
		
		//transition from WaitZ3Ready to Recovering / MoveForward
		IF bStopRequest THEN 
			eNewStep := E_Z2_Step.Recovering;
		ELSIF stStatus.stZ3.eStep = E_Z3_Step.Ready THEN
			eNewStep := E_Z2_Step.MoveForward; 
		END_IF; 	
	
		// exit action
		IF eNewStep <> E_Z2_Step.NoStep THEN
			;
		END_IF;
			
	// MoveForward
    E_Z2_Step.MoveForward :
		// entry action
		IF NOT bEntryact THEN
			bErr := FALSE;
			bEntryact := TRUE;
		END_IF;
		
		//body
		bQ1 := FALSE;
		bQ2 := NOT(bI1);
		
		//transition from MoveForward to MoveBackward
		IF (fbRtI1.Q) THEN
			eNewStep := E_Z2_Step.MoveBackward; 
		END_IF;
		
		// exit action
		IF eNewStep <> E_Z2_Step.NoStep THEN
			;
		END_IF;
	
	// MoveBackward
    E_Z2_Step.MoveBackward :
		// entry action
		IF NOT bEntryact THEN
			bErr := FALSE;
			bEntryact := TRUE;
		END_IF;
		
		//body
		bQ1 :=  NOT(bI2);
		bQ2 := FALSE;
		
		//transition from MoveBackward to Done
		IF (fbRtI2.Q) THEN
			eNewStep := E_Z2_Step.Done; 
		END_IF;
		
		// exit action
		IF eNewStep <> E_Z2_Step.NoStep THEN
			;
		END_IF;
	
   // Done
    E_Z2_Step.Done :
		// entry action
		IF NOT bEntryact THEN
			bErr := FALSE;
			bEntryact := TRUE;
		END_IF;
		
		//body
		bQ1 :=  FALSE;
		bQ2 :=  FALSE;
		
		//transition from MoveBackward to Done
		eNewStep := E_Z2_Step.Ready; 
		
		// exit action
		IF eNewStep <> E_Z2_Step.NoStep THEN
			;
		END_IF;
		
	ELSE
			eNewstep :=  E_Z2_Step.NeOrError;
			stStatus.stZ2.eErrorStep :=  E_Z2_Step.Unknown;			
			stStatus.stZ2.nErrorId := 16#0002_9999;
	END_CASE 
	
	(* call FBs *)
	
	(* tempo di permanenza nello step *)
	fbTonStep(IN := (eNewstep =  E_Z2_Step.NoStep), PT := T#500H);
	stStatus.stZ2.tStepTime := fbTonStep.ET;	
END_IF

END_FUNCTION_BLOCK

// ---- FSM/Z3/FB_Z3_FSM.TcPOU
FUNCTION_BLOCK FB_Z3_FSM
VAR_INPUT
	bEnable		:	BOOL;
	bAck		:	BOOL;
	bStop		:	BOOL;
	bI6			:	BOOL;
	stParams	:	ST_Z3_Params;	
END_VAR
VAR_IN_OUT
	stStatus	:	ST_FSM_Status;
END_VAR
VAR_OUTPUT
	// Digital Outputs
	bQ6			:	BOOL;
	bQ7			:	BOOL;	
	bErr		:	BOOL;
END_VAR

VAR
	// FSM internal variables
	bInitialized	:	BOOL;
	eNewstep		:	E_Z3_Step;
	bEntryact		:	BOOL;
	fbTonStep		:	TON;
	
	fbRtStop		:	R_TRIG;
	fbRtI6			:	R_TRIG;
	bStopRequest	:	BOOL;

	// object on conveyor
	bConveyorLoaded	:	BOOL;	
END_VAR

IF NOT bInitialized THEN
	eNewstep :=  E_Z3_Step.NoStep;
	stStatus.stZ3.eStep :=  E_Z3_Step.NeOrError;
	bEntryact := FALSE;
	bInitialized := TRUE;	
	bErr := FALSE;
	stStatus.stZ3.eErrorStep :=  E_Z3_Step.NoStep;	
	stStatus.stZ3.nErrorId := 0;	
ELSE
	(* fronti *)
	fbRtStop(CLK:= bStop);	
	fbRtI6(CLK := bI6);
	
	(* richieste *)
	IF fbRtStop.Q THEN
		bStopRequest := TRUE;
	END_IF; 

	(* disabilitata o avaria *)
	IF NOT bEnable THEN
		eNewstep := E_Z3_Step.NeOrError;
	END_IF;
	
	(* aggiornamento dello stato *)
	IF eNewstep <>  E_Z3_Step.NoStep THEN
		stStatus.stZ3.eStep := eNewstep;
		eNewstep :=  E_Z3_Step.NoStep;
		bEntryact := FALSE;
	END_IF;	
	
	(* switch - case della MSF *)
	CASE stStatus.stZ3.eStep OF
		
		// NeOrError ---------------------------------
		E_Z3_Step.NeOrError :
			// on entry action
			IF NOT bEntryact THEN
				bErr := TRUE;
				bEntryact := TRUE;
			END_IF
			
			// body
			bQ6 := FALSE;
			bQ7 := FALSE;					
			
			// next state transition
			IF bEnable THEN
				IF bAck THEN
					eNewStep := E_Z3_Step.Recovering;
				END_IF
			END_IF
		
			// on exit action
			IF eNewStep <> E_Z3_Step.NoStep THEN
				stStatus.stZ3.nErrorId := 0;
				stStatus.stZ3.eErrorStep := E_Z3_Step.NoStep;
			END_IF
	
		// Recovering ---------------------------------			
		E_Z3_Step.Recovering :
			// on entry action
			IF NOT bEntryact THEN
				bErr := FALSE;				
				bEntryact := TRUE;
			END_IF
			
			// body	
			bQ6 := FALSE;
			bQ7 := FALSE;

			// next state transition
			IF bEnable THEN
				IF (stStatus.stZ3.tStepTime > stParams.tRecovering) THEN
					eNewStep := E_Z3_Step.Stop;
				END_IF				
			END_IF
			
			// on exit action
			IF eNewStep <> E_Z3_Step.NoStep THEN
				;
			END_IF			
			
		// Stop ---------------------------------------
		E_Z3_Step.Stop :
			// on entry action
			IF NOT bEntryact THEN
				bErr:= FALSE;				
				bStopRequest := FALSE;
				bConveyorLoaded := FALSE;
				bEntryact := TRUE;
			END_IF
			
			// body	
			bQ6 := FALSE;
			bQ7 := FALSE;
			
			// next state transition
			IF bEnable THEN
				IF (stStatus.stZ3.tStepTime > stParams.tStopDelay) THEN
					eNewStep := E_Z3_Step.Ready;
				END_IF
			END_IF
			
			// on exit action
			IF eNewStep <> E_Z3_Step.NoStep THEN
				;
			END_IF
			
		// Ready ---------------------------------------
		E_Z3_Step.Ready :
			// on entry action
			IF NOT bEntryact THEN
				bErr:= FALSE;				
				bConveyorLoaded := FALSE;
				bEntryact := TRUE;
			END_IF
			
			// body	
			bQ6 := FALSE;
			bQ7 := FALSE;

			// next state transition
			IF bStopRequest THEN 
				eNewStep := E_Z3_Step.Recovering;
			ELSIF stStatus.stZ2.eStep=E_Z2_Step.WaitZ3Ready THEN
				eNewStep := E_Z3_Step.MoveToMill;
			END_IF
			
			// on exit action
			IF eNewStep <> E_Z3_Step.NoStep THEN
				;
			END_IF
			
			// MoveToMill ---------------------------------------
		E_Z3_Step.MoveToMill :
			// on entry action
			IF NOT bEntryact THEN
				bErr:= FALSE;				
				bConveyorLoaded := TRUE;
				bEntryact := TRUE;
			END_IF
			
			// body	
			bQ6 := NOT(bI6);
			bQ7 := FALSE;
	
			// next state transition
			IF bStopRequest THEN 
				eNewStep := E_Z3_Step.Recovering;
			ELSIF bI6 THEN
				eNewStep := E_Z3_Step.Milling;
			END_IF
			
			// on exit action
			IF eNewStep <> E_Z3_Step.NoStep THEN
				;
			END_IF
						

		// Milling ---------------------------------------
		E_Z3_Step.Milling :
			// on entry action
			IF NOT bEntryact THEN
				bErr:= FALSE;
				bConveyorLoaded := TRUE;
				bEntryact := TRUE;
			END_IF
			
			// body	
			bQ6 := FALSE;
			bQ7 := TRUE;
			
			// next state transition
			IF stStatus.stZ3.tStepTime > stParams.tMilling THEN 
				eNewStep := E_Z3_Step.WaitZ4Ready;
			END_IF
			
			// on exit action
			IF eNewStep <> E_Z3_Step.NoStep THEN
				;
			END_IF
			
		// WaitZ4Ready ---------------------------------------
		E_Z3_Step.WaitZ4Ready :
			// on entry action
			IF NOT bEntryact THEN
				bErr:= FALSE;
				bConveyorLoaded := TRUE;
				bEntryact := TRUE;
			END_IF
			
			// body	
			bQ6 := FALSE;
			bQ7 := FALSE;
			
			// next state transition
			IF stStatus.stZ4.eStep=E_Z4_Step.Ready THEN 
				eNewStep := E_Z3_Step.MoveToZ4;
			END_IF
			
			// on exit action
			IF eNewStep <> E_Z3_Step.NoStep THEN
				;
			END_IF
			
		// MoveToZ4 ---------------------------------------
		E_Z3_Step.MoveToZ4 :
			// on entry action
			IF NOT bEntryact THEN
				bErr:= FALSE;
				bConveyorLoaded := TRUE;
				bEntryact := TRUE;
			END_IF
			
			// body	
			bQ6 := TRUE;
			bQ7 := FALSE;
			
			// next state transition
			IF stStatus.stZ3.tStepTime > stParams.tDelayToZ4 THEN 
				eNewStep := E_Z3_Step.Done;
			END_IF
			
			// on exit action
			IF eNewStep <> E_Z3_Step.NoStep THEN
				;
			END_IF
			
		// Done ---------------------------------------
		E_Z3_Step.Done :
			// on entry action
			IF NOT bEntryact THEN
				bErr:= FALSE;
				bConveyorLoaded := FALSE;
				bEntryact := TRUE;
			END_IF
			
			// body	
			bQ6 := FALSE;
			bQ7 := FALSE;
			
			// next state transition
			eNewStep := E_Z3_Step.Ready;
			
			
			// on exit action
			IF eNewStep <> E_Z3_Step.NoStep THEN
				;
			END_IF
			
	ELSE
			eNewstep :=  E_Z3_Step.NeOrError;
			stStatus.stZ3.eErrorStep :=  E_Z3_Step.Unknown;			
			stStatus.stZ3.nErrorId := 16#0003_9999;	
	END_CASE
	
	(* call FBs *)
	
	(* tempo di permanenza nello step *)
	fbTonStep(IN := (eNewstep =  E_Z3_Step.NoStep), PT := T#500H);
	stStatus.stZ3.tStepTime := fbTonStep.ET;	
	
END_IF

END_FUNCTION_BLOCK

// ---- FSM/Z4/FB_Z4_FSM.TcPOU
FUNCTION_BLOCK FB_Z4_FSM
VAR_INPUT
	bEnable		:	BOOL;
	bAck		:	BOOL;
	bStop		:	BOOL;
	bI8			:	BOOL;
	stParams	:	ST_Z4_Params;	
END_VAR
VAR_IN_OUT
	stStatus	:	ST_FSM_Status;	
END_VAR
VAR_OUTPUT
	// Digital Outputs
	bQ8			:	BOOL;
	bQ9			:	BOOL;	
	bErr		:	BOOL;
END_VAR
VAR
	// FSM internal variables
	bInitialized	:	BOOL;
	eNewstep		:	E_Z4_Step;
	bEntryact		:	BOOL;
	fbTonStep		:	TON;
	
	fbRtStop		:	R_TRIG;
	fbRtI8			:	R_TRIG;
	bStopRequest	:	BOOL;	
	bConveyorLoaded :   BOOL;
END_VAR

IF NOT bInitialized THEN
	eNewstep :=  E_Z4_Step.NoStep;
	stStatus.stZ4.eStep :=  E_Z4_Step.NeOrError;
	bEntryact := FALSE;
	bInitialized := TRUE;	
	bErr := FALSE;
	stStatus.stZ4.eErrorStep :=  E_Z4_Step.NoStep;	
	stStatus.stZ4.nErrorId := 0;	
ELSE
	(* fronti *)
	fbRtStop(CLK:= bStop);	
	fbRtI8(CLK := bI8);
	
	(* richieste *)
	IF fbRtStop.Q THEN
		bStopRequest := TRUE;
	END_IF; 

	(* disabilitata o avaria *)
	IF NOT bEnable THEN
		eNewstep := E_Z4_Step.NeOrError;
	END_IF;
	
	(* aggiornamento dello stato *)
	IF eNewstep <>  E_Z4_Step.NoStep THEN
		stStatus.stZ4.eStep := eNewstep;
		eNewstep :=  E_Z4_Step.NoStep;
		bEntryact := FALSE;
	END_IF
	
	(* Guasto e Rispristino *)
	IF stStatus.bFailure THEN
		eNewStep :=	E_Z4_Step.NeOrError;
	END_IF

	(* switch - case della MSF *)
	CASE stStatus.stZ4.eStep OF
		
	// NeOrError ---------------------------------			
	E_Z4_Step.NeOrError :
		// on entry action
		IF NOT bEntryact THEN
			bErr := TRUE;
			bEntryact := TRUE;
		END_IF
		
		// body
		bQ8 := FALSE;
		bQ9 := FALSE;			
			
		// next state transition
		IF bEnable THEN
			IF bAck THEN
				eNewStep := E_Z4_Step.Recovering;
			END_IF
		END_IF
		
		// on exit action
		IF eNewStep <> E_Z4_Step.NoStep THEN
			stStatus.stZ4.nErrorId := 4;
			stStatus.stZ4.eErrorStep := E_Z4_Step.NoStep;
		END_IF
	
	// Recovering ---------------------------------			
	E_Z4_Step.Recovering :
		// on entry action
		IF NOT bEntryact THEN
			bErr := FALSE;			
			bEntryact := TRUE;
		END_IF
			
		// body	
		bQ8 := FALSE;
		bQ9 := FALSE;
		
		// next state transition
		IF bEnable THEN
			eNewStep := E_Z4_Step.Stop;			
		END_IF
		
		// on exit action
		IF eNewStep <> E_Z4_Step.NoStep THEN
			;
		END_IF			
			
	// Stop ---------------------------------------
	E_Z4_Step.Stop :
		// on entry action
		IF NOT bEntryact THEN
			bStopRequest := FALSE;
			bErr:= FALSE;				
			bEntryact := TRUE;
		END_IF
			
		// body	
		bQ8 := FALSE;
		bQ9 := FALSE;
			
		// next state transition
		IF (stStatus.stZ4.tStepTime > stParams.tStopDelay) THEN
			eNewStep := E_Z4_Step.Ready;
		END_IF

		// on exit action
		IF eNewStep <> E_Z4_Step.NoStep THEN
			;
		END_IF
			
	// Ready ---------------------------------------
	E_Z4_Step.Ready :
		// on entry action
		IF NOT bEntryact THEN
			bErr:= FALSE;
			bEntryact := TRUE;
		END_IF
			
		// body	
		bQ8 := FALSE;
		bQ9 := FALSE;
						
		// next state transition
		IF bStopRequest THEN 
			eNewStep := E_Z4_Step.Recovering;
		ELSIF stStatus.stZ3.eStep = E_Z3_Step.WaitZ4Ready THEN
			eNewStep := E_Z4_Step.MoveToDrill;
		END_IF
		
		// on exit action
		IF eNewStep <> E_Z4_Step.NoStep THEN
			;
		END_IF
			
	// MoveToDrill ---------------------------------------
	E_Z4_Step.MoveToDrill :
		// on entry action
		IF NOT bEntryact THEN
			bErr:= FALSE;
			bEntryact := TRUE;
		END_IF
			
		// body	
		bQ8 := NOT(bI8);
		bQ9 := FALSE;
			
		// next state transition
		IF bStopRequest THEN 
			eNewStep := E_Z4_Step.Recovering;
		ELSIF fbRtI8.Q THEN
			eNewStep := E_Z4_Step.Drilling;
		END_IF
			
		// on exit action
		IF eNewStep <> E_Z4_Step.NoStep THEN
			;
		END_IF
						
	// Drilling ---------------------------------------
	E_Z4_Step.Drilling :
		// on entry action
		IF NOT bEntryact THEN
			bErr:= FALSE;
			bEntryact := TRUE;
		END_IF
			
		// body	
		bQ8 := FALSE;
		bQ9 := TRUE;
			
		// next state transition
		IF stStatus.stZ4.tStepTime > stParams.tDrilling THEN 
			eNewStep := E_Z4_Step.WaitZ5Ready;
		END_IF
			
		// on exit action
		IF eNewStep <> E_Z4_Step.NoStep THEN
			;
		END_IF
			
	// WaitZ5Ready ---------------------------------------
	E_Z4_Step.WaitZ5Ready :
		// on entry action
		IF NOT bEntryact THEN
			bErr:= FALSE;
			bEntryact := TRUE;
		END_IF
			
		// body	
		bQ8 := FALSE;
		bQ9 := FALSE;

		// next state transition
		IF stStatus.stZ5.eStep=E_Z5_Step.Ready THEN 
			eNewStep := E_Z4_Step.MoveToZ5;
		END_IF
			
		// on exit action
		IF eNewStep <> E_Z4_Step.NoStep THEN
			;
		END_IF
			
	// MoveToZ5 ---------------------------------------
	E_Z4_Step.MoveToZ5 :
		// on entry action
		IF NOT bEntryact THEN
			bErr:= FALSE;
			bEntryact := TRUE;
		END_IF
		
		// body	
		bQ8 := TRUE;
		bQ9 := FALSE;

		// next state transition
		IF stStatus.stZ4.tStepTime > stParams.tDelayToZ5 THEN 
			eNewStep := E_Z4_Step.Done;
		END_IF
		
		// on exit action
		IF eNewStep <> E_Z4_Step.NoStep THEN
			;
		END_IF
			
	// Done ---------------------------------------
	E_Z4_Step.Done :
		// on entry action
		IF NOT bEntryact THEN
			bErr:= FALSE;
			bEntryact := TRUE;
		END_IF
			
		// body	
		bQ8 := FALSE;
		bQ9 := FALSE;
	
		// next state transition	
		eNewStep := E_Z4_Step.Ready;
		
		// on exit action
		IF eNewStep <> E_Z4_Step.NoStep THEN
			;
		END_IF

	ELSE
			eNewstep :=  E_Z4_Step.NeOrError;
			stStatus.stZ4.eErrorStep :=  E_Z4_Step.Unknown;			
			stStatus.stZ4.nErrorId := 16#0004_9999;	
	END_CASE
	
	(* call FBs *)
	
	(* tempo di permanenza nello step *)
	fbTonStep(IN := (eNewstep =  E_Z4_Step.NoStep), PT := T#500H);
	stStatus.stZ4.tStepTime := fbTonStep.ET;	
	
END_IF

END_FUNCTION_BLOCK

// ---- FSM/Z5/FB_Z5_FSM.TcPOU
FUNCTION_BLOCK FB_Z5_FSM
VAR_INPUT
	bEnable		:	BOOL;
	bAck		:	BOOL;
	bStop		:	BOOL;
	bI3			:	BOOL;
	bI4			:	BOOL;
	stParams	:	ST_Z5_Params;	
END_VAR
VAR_IN_OUT
	stStatus	:	ST_FSM_Status;	
END_VAR
VAR_OUTPUT
	// Digital Outputs
	bQ3			:	BOOL;
	bQ4			:	BOOL;	
	bErr		:	BOOL;
END_VAR
VAR
	// FSM internal variables
	bInitialized	:	BOOL;
	eNewstep		:	E_Z5_Step;
	bEntryact		:	BOOL;
	fbTonStep		:	TON;
	
	fbRtStop		:	R_TRIG;
	fbRtI3			:	R_TRIG;
	fbRtI4			:	R_TRIG;
	bStopRequest	:	BOOL;	
END_VAR

IF NOT bInitialized THEN
	eNewstep :=  E_Z5_Step.NoStep;
	stStatus.stZ5.eStep :=  E_Z5_Step.NeOrError;
	bEntryact := FALSE;
	bInitialized := TRUE;	
	bErr := FALSE;
	stStatus.stZ5.eErrorStep :=  E_Z5_Step.NoStep;	
	stStatus.stZ5.nErrorId := 0;	
ELSE
	(* fronti *)
	fbRtStop(CLK:= bStop);	
	fbRtI3(CLK := bI3);
	fbRtI4(CLK := bI4);
	
	(* richieste *)
	IF fbRtStop.Q THEN
		bStopRequest := TRUE;
	END_IF; 

	(* disabilitata o avaria *)
	IF NOT bEnable THEN
		eNewstep := E_Z5_Step.NeOrError;
	END_IF;
	
	(* aggiornamento dello stato *)
	IF eNewstep <>  E_Z5_Step.NoStep THEN
		stStatus.stZ5.eStep := eNewstep;
		eNewstep :=  E_Z5_Step.NoStep;
		bEntryact := FALSE;
	END_IF;	
	
	(* switch - case della MSF *)
	CASE stStatus.stZ5.eStep OF
	
	// NeOrError -----------------------------------------
	E_Z5_Step.NeOrError :
		// entry action
		IF NOT bEntryact THEN
			bErr := TRUE;
			bEntryact := TRUE;
		END_IF
		
		// body
		bQ3 := FALSE;
		bQ4 := FALSE;
		
		// transition from NeOrError to Recovering
		IF (bEnable AND bAck) THEN
			eNewStep := E_Z5_Step.Recovering;
		END_IF
		
		// exit action
		IF eNewStep <> E_Z5_Step.NoStep THEN
			stStatus.stZ5.nErrorID := 5;
			stStatus.stZ5.eErrorStep := E_Z5_Step.NoStep;
		END_IF	

	// Recovering -----------------------------------------
	E_Z5_Step.Recovering :
		// entry action
		IF NOT bEntryact THEN
			bErr := FALSE;
			bEntryact := TRUE;
		END_IF
		
		// body
		bQ3 := NOT(bI4);
		bQ4 := FALSE;
		
		// transition from Recovering to Stop
		IF fbRtI4.Q THEN
			eNewStep := E_Z5_Step.Stop;
		END_IF
		
		// exit action
		IF eNewStep <> E_Z5_Step.NoStep THEN
			;
		END_IF	

	// Stop -----------------------------------------
	E_Z5_Step.Stop :
		// entry action
		IF NOT bEntryact THEN
			bErr := FALSE;
			bEntryact := TRUE;
		END_IF
		
		// body
		bQ3 := FALSE;
		bQ4 := FALSE;
		
		// transition from Stop to Ready
		IF stStatus.stZ5.tStepTime > stParams.tStopDelay THEN
			eNewStep := E_Z5_Step.Ready;
		END_IF
		
		// exit action
		IF eNewStep <> E_Z5_Step.NoStep THEN
			;
		END_IF	

	// Ready -----------------------------------------
	E_Z5_Step.Ready :
		// entry action
		IF NOT bEntryact THEN
			bErr := FALSE;
			bEntryact := TRUE;
		END_IF
		
		// body
		bQ3 := FALSE;
		bQ4 := FALSE;
		
		// transition from Ready to Recovering / WaitZ6Ready
		IF bStopRequest THEN
			eNewStep := E_Z5_Step.Recovering;
		ELSE
			IF stStatus.stZ4.eStep = E_Z4_Step.WaitZ5Ready THEN
				eNewStep := E_Z5_Step.WaitZ6Ready;
			END_IF			
		END_IF

		// exit action
		IF eNewStep <> E_Z5_Step.NoStep THEN
			;
		END_IF	
		
	// WaitZ6Ready -----------------------------------------
	E_Z5_Step.WaitZ6Ready :
		// entry action
		IF NOT bEntryact THEN
			bErr := FALSE;
			bEntryact := TRUE;
		END_IF
		
		// body
		bQ3 := FALSE;
		bQ4 := FALSE;
		
		// transition from WaitZ6Ready to Recovering / MoveForward
		IF bStopRequest THEN
			eNewStep := E_Z5_Step.Recovering;
		ELSE
			IF stStatus.stZ6.eStep = E_Z6_Step.Ready THEN
				eNewStep := E_Z5_Step.MoveForward;
			END_IF			
		END_IF

		// exit action
		IF eNewStep <> E_Z5_Step.NoStep THEN
			;
		END_IF	
	
	// MoveForward -----------------------------------------
	E_Z5_Step.MoveForward :
		// entry action
		IF NOT bEntryact THEN
			bErr := FALSE;
			bEntryact := TRUE;
		END_IF
		
		// body
		bQ3 := FALSE;
		bQ4 := NOT(bI3);
		
		// transition from MoveForward to MoveBackward
		IF fbRtI3.Q THEN
			eNewStep := E_Z5_Step.MoveBackward;			
		END_IF

		// exit action
		IF eNewStep <> E_Z5_Step.NoStep THEN
			;
		END_IF
		
	// MoveBackward -----------------------------------------
	E_Z5_Step.MoveBackward :
		// entry action
		IF NOT bEntryact THEN
			bErr := FALSE;
			bEntryact := TRUE;
		END_IF
		
		// body
		bQ3 := NOT(bI4);
		bQ4 := FALSE;
		
		// transition from MoveBackward to Done
		IF fbRtI4.Q THEN
			eNewStep := E_Z5_Step.Done;			
		END_IF

		// exit action
		IF eNewStep <> E_Z5_Step.NoStep THEN
			;
		END_IF	

	// Done -----------------------------------------
	E_Z5_Step.Done:
		// entry action
		IF NOT bEntryact THEN
			bErr := FALSE;
			bEntryact := TRUE;
		END_IF
		
		// body
		bQ3 := FALSE;
		bQ4 := FALSE;
		
		// transition from Done to Ready
		eNewStep := E_Z5_Step.Ready;			

		// exit action
		IF eNewStep <> E_Z5_Step.NoStep THEN
			;
		END_IF		
		
	ELSE
			eNewstep :=  E_Z5_Step.NeOrError;
			stStatus.stZ5.eErrorStep :=  E_Z5_Step.Unknown;			
			stStatus.stZ5.nErrorId := 16#0005_9999;	
	END_CASE
	
	(* call FBs *)
	
	(* tempo di permanenza nello step *)
	fbTonStep(IN := (eNewstep =  E_Z5_Step.NoStep), PT := T#500H);
	stStatus.stZ5.tStepTime := fbTonStep.ET;	
	
END_IF

END_FUNCTION_BLOCK

// ---- FSM/Z6/FB_Z6_FSM.TcPOU
FUNCTION_BLOCK FB_Z6_FSM
VAR_INPUT
	bEnable		:	BOOL;
	bAck		:	BOOL;
	bStop		:	BOOL;
	bI9			:	BOOL;
	stParams	:	ST_Z6_Params;	
END_VAR
VAR_IN_OUT
	stStatus	:	ST_FSM_Status;	
END_VAR
VAR_OUTPUT
	// Digital Outputs
	bQ10		:	BOOL;
	bErr		:	BOOL;
END_VAR
VAR
	// FSM internal variables
	bInitialized	:	BOOL;
	eNewstep		:	E_Z6_Step;
	bEntryact		:	BOOL;
	fbTonStep		:	TON;
	
	fbRtStop		:	R_TRIG;
	fbRtI9			:	R_TRIG;
	bStopRequest	:	BOOL;	
END_VAR

IF NOT bInitialized THEN
	eNewstep :=  E_Z6_Step.NoStep;
	stStatus.stZ6.eStep :=  E_Z6_Step.NeOrError;
	bEntryact := FALSE;
	bInitialized := TRUE;	
	bErr := FALSE;
	stStatus.stZ6.eErrorStep :=  E_Z6_Step.NoStep;	
	stStatus.stZ6.nErrorId := 0;	
ELSE
	(* fronti *)
	fbRtStop(CLK:= bStop);	
	fbRtI9(CLK := bI9);
	
	(* richieste *)
	IF fbRtStop.Q THEN
		bStopRequest := TRUE;
	END_IF; 

	(* disabilitata o avaria *)
	IF NOT bEnable THEN
		eNewstep := E_Z6_Step.NeOrError;
	END_IF;
	
	(* aggiornamento dello stato *)
	IF eNewstep <>  E_Z6_Step.NoStep THEN
		stStatus.stZ6.eStep := eNewstep;
		eNewstep :=  E_Z6_Step.NoStep;
		bEntryact := FALSE;
	END_IF;	
	
	IF stStatus.bFailure THEN
		eNewstep := E_Z6_Step.NeOrError;
	END_IF
	
	(* switch - case della MSF *)
	CASE stStatus.stZ6.eStep OF

	// STOP ------------------------------------------
	E_Z6_Step.Stop	:
		//entry act
		IF NOT bEntryact THEN
			bErr := FALSE;
			bEntryact := TRUE;
		END_IF
		
		// Body
		bQ10 := FALSE;
		
		// transition from Stop to Ready
		IF(stStatus.stZ6.tStepTime > stParams.tStopDelay) THEN
			eNewStep := E_Z6_Step.Ready;
		END_IF
	
		// exit action
		IF eNewStep <> E_Z6_Step.NoStep THEN
			;
		END_IF		
		
	// READY ------------------------------------------
	E_Z6_Step.Ready:
		//entry act
		IF NOT bEntryact THEN
			bErr := FALSE;
			bEntryact := TRUE;
		END_IF
		
		// Body		
		bQ10 := FALSE;
		
		// transition from Ready to Loading / Recovering
		IF bStopRequest THEN
			eNewStep := E_Z6_Step.Recovering;
		ELSE
			IF (stStatus.stZ5.eStep = E_Z5_Step.WaitZ6Ready) THEN
				eNewStep := E_Z6_Step.Loading;
			END_IF
		END_IF		
	
		// exit action
		IF eNewStep <> E_Z6_Step.NoStep THEN
			;
		END_IF	
	
	// LOADING ------------------------------------------
	E_Z6_Step.Loading:
		//entry act
		IF NOT bEntryact THEN
			bErr := FALSE;
			bEntryact := TRUE;
		END_IF
		
		// Body	
		bQ10 := TRUE;
		
		// transition from Loading to Recovering / WaitUnloading
		IF bStopRequest THEN
			eNewStep := E_Z6_Step.Recovering;
		ELSE
			IF fbrtI9.Q THEN
				eNewStep := E_Z6_Step.WaitUnloading;
			END_IF
		END_IF
	
		// exit action
		IF eNewStep <> E_Z6_Step.NoStep THEN
			;
		END_IF	
	
	// WAIT_UNLOADING ------------------------------------------
	E_Z6_Step.WaitUnloading	:
		//entry act
		IF NOT bEntryact THEN
			bErr := FALSE;
			bEntryact := TRUE;
		END_IF
		
		// Body		
		bQ10	:=	FALSE;

		// transition from WaitUnloading to Done	
		IF NOT(bI9) THEN
			eNewStep := E_Z6_Step.Done;
		END_IF
	
		// exit action
		IF eNewStep <> E_Z6_Step.NoStep THEN
			;
		END_IF	
	
	// DONE	
	E_Z6_Step.Done	:
		//entry act
		IF NOT bEntryact THEN
			bErr := FALSE;
			bEntryact := TRUE;
		END_IF
		
		// Body		
		bQ10 := FALSE;

		// transition from Done to Ready	
		eNewStep := E_Z6_Step.Ready;
	
		// exit action
		IF eNewStep <> E_Z6_Step.NoStep THEN
			;
		END_IF	
	
	// NEORERROR ------------------------------------------
	E_Z6_Step.NeOrError:
		//entry act	
		IF NOT bEntryact THEN
			bErr := TRUE;
			bEntryact := TRUE;
		END_IF
		
		// Body		
		bQ10	:=	FALSE;

		// transition from NeOrError to Recovering	
		IF bEnable THEN
			IF bAck THEN
				eNewStep := E_Z6_Step.Recovering;
			END_IF
		END_IF
	
		//exit act
		IF eNewStep <> E_Z6_Step.NoStep THEN
			stStatus.stZ6.nErrorId := 0;
			stStatus.stZ6.eErrorStep := E_Z6_Step.NoStep;
		END_IF	
	
	// RECOVERING ------------------------------------------
	E_Z6_Step.Recovering:
		//entry act	
		IF NOT bEntryact THEN
			bErr := FALSE;
			bEntryact := TRUE;
		END_IF
		
		// Body	
		bQ10 := FALSE;

		// transition from Recovering to Stop	
		IF bEnable THEN
			IF NOT(stStatus.bFailure) THEN
				eNewStep := E_Z6_Step.Stop;
			END_IF				
		END_IF
	
		// exit action
		IF eNewStep <> E_Z6_Step.NoStep THEN
			;
		END_IF
	
	ELSE
			eNewstep :=  E_Z6_Step.NeOrError;
			stStatus.stZ6.eErrorStep :=  E_Z6_Step.Unknown;			
			stStatus.stZ6.nErrorId := 16#0006_9999;	
	END_CASE
	
	(* call FBs *)
	
	(* tempo di permanenza nello step *)
	fbTonStep(IN := (eNewstep =  E_Z6_Step.NoStep), PT := T#500H);
	stStatus.stZ6.tStepTime := fbTonStep.ET;	
	
END_IF

END_FUNCTION_BLOCK

// ---- FSM/Coordinator/FCs/FC_AllStopped.TcPOU
FUNCTION FC_AllStopped : BOOL
VAR_INPUT
	stStatus	:	ST_FSM_Status;
END_VAR
VAR
END_VAR

FC_AllStopped := (stStatus.stZ1.eStep = E_Z1_Step.Stop) AND
                 (stStatus.stZ2.eStep = E_Z2_Step.Stop) AND
                 (stStatus.stZ3.eStep = E_Z3_Step.Stop) AND	
                 (stStatus.stZ4.eStep = E_Z4_Step.Stop) AND
                 (stStatus.stZ5.eStep = E_Z5_Step.Stop) AND	
                 (stStatus.stZ6.eStep = E_Z6_Step.Stop);

END_FUNCTION

// ---- POUs/MAIN.TcPOU
PROGRAM MAIN
VAR
	
	bInitialized		:	BOOL;
	bPLCTaskRunning		:	BOOL;
	
	fbGetCurTaskIndex	:	GETCURTASKINDEX;		
	tTaskCycleTime		:	UDINT;				// CycleTime is expressed in microseconds
	tTaskExecTime		:	UDINT;				// task execution time expressed in microseconds
	tTaskMaxExecTime	:	UDINT;				// maximum task execution time expressed in microseconds
	
	(* instantiate the main state machine FB_FSM_Main *)
	fbFsm				:	FB_FSM_Main;
	
	(* Local variables *)
	stRawIn				:	ST_FSM_RawIn;
	stIn				:	ST_FSM_In;
	stRawOut			:	ST_FSM_RawOut;
	stOut				:	ST_FSM_Out;
	stCtrl				:	ST_FSM_Ctrl;
	stStatus			:	ST_FSM_Status;
	
END_VAR

IF NOT bInitialized THEN
	
	// Get the Cycle Time of the task to which this PRG is assigned (it will then be shared with the State Machine)
	fbGetCurTaskIndex();
	tTaskCycleTime := _TaskInfo[fbGetCurTaskIndex.index].CycleTime / 10;	// CycleTime is expressed in multiples of 100ns
	bInitialized := TRUE;
	
ELSE
	
	(* task time *)
	tTaskExecTime := _TaskInfo[fbGetCurTaskIndex.index].LastExecTime / 10;		// ExecTime is expressed in multiples of 100ns
	IF tTaskExecTime > tTaskMaxExecTime THEN
			tTaskMaxExecTime := tTaskExecTime;
	END_IF;	
	
	(* execute main state machine *)
	fbFsm(
	bEnable:= TRUE, 
	tTaskCycleTime:= tTaskExecTime, 
	nId:= 0, 
	bHwError:= FALSE, 
	stRawIn:= stRawIn, 
	stIn:= stIn, 
	stRawOut:= stRawOut, 
	stOut:= stOut, 
	stCtrl:= stCtrl, 
	stStatus:= stStatus);	
	
	(* system signal *)
	bPLCTaskRunning := TRUE;
END_IF

END_PROGRAM
